// TIA Portal V20 export
DATA_BLOCK "DB_Simulation"   // DB99
// stored: InstanceOfName FB_Simulation, InstanceOfType FB
"FB_Simulation"
   // VAR
   //    sExtLoadUnloadTimer1 : TON_TIME;
   //    sExtLoadUnloadTimer2 { S7_SetPoint := 'True'} : TON_TIME;
   //    sBwLoadUnloadTimer1 { S7_SetPoint := 'True'} : TON_TIME;
   //    sBwLoadUnloadTimer2 { S7_SetPoint := 'True'} : TON_TIME;
   //    sTON_UndrilledGripperFull { S7_SetPoint := 'True'} : TON_TIME;
   //    sTON_UndrilledFixture { S7_SetPoint := 'True'} : TON_TIME;
   //    sTON_DrilledFixture { S7_SetPoint := 'True'} : TON_TIME;
   //    sTON_ResetBit { S7_SetPoint := 'True'} : TON_TIME;
   //    sSeqRun { S7_SetPoint := 'True'} : Bool;
   //    sTON_CloseDrilledGripper_1 { S7_SetPoint := 'True'} : TON_TIME;
   //    sTONCloseFixture { S7_SetPoint := 'True'} : TON_TIME;
   //    sTONOpenFixture { S7_SetPoint := 'True'} : TON_TIME;
   //    sTONOpenFixture1 { S7_SetPoint := 'True'} : TON_TIME;
   //    sTON_CloseDrilledGripper { S7_SetPoint := 'True'} : TON_TIME;
   //    sTON_WorkinProgress { S7_SetPoint := 'True'} : TON_TIME;
   //    sTON_OpenUndrilledGripper { S7_SetPoint := 'True'} : TON_TIME;
   //    sRT_NC_Mode { S7_SetPoint := 'True'} : R_TRIG;
   //    sStep { S7_SetPoint := 'True'} : Array[0..15] of Bool;
   //    sRT_DrillingFinished : R_TRIG;
   //    "sTON_No MCodes" { S7_SetPoint := 'True'} : TON_TIME;
   //    sRT_TONMCodes { S7_SetPoint := 'True'} : R_TRIG;
   //    sRT_FIXLoading { S7_SetPoint := 'True'} : R_TRIG;
   //    sRT_FIXblowing { S7_SetPoint := 'True'} : R_TRIG;
   //    sRT_MemoLoaderStart { S7_SetPoint := 'True'} : R_TRIG;
   //    sRT_Sh1_ExtLoadUnloadDone { S7_SetPoint := 'True'} : R_TRIG;
   //    sRT_Sh2_ExtLoadUnloadDone { S7_SetPoint := 'True'} : R_TRIG;
   // END_VAR
BEGIN
END_DATA_BLOCK
